(* IEC 61131-3 sources: CBasicModel/PLC/build, 2 files *)

(* ---- plc.st ---- *)
TYPE
  LOGLEVEL : (CRITICAL, WARNING, INFO, DEBUG) := INFO;
END_TYPE

FUNCTION_BLOCK LOGGER
  VAR_INPUT
    TRIG : BOOL;
    MSG : STRING;
    LEVEL : LOGLEVEL := INFO;
  END_VAR
  VAR
    TRIG0 : BOOL;
  END_VAR

  IF TRIG AND NOT TRIG0 THEN
  {{
   LogMessage(GetFbVar(LEVEL),(char*)GetFbVar(MSG, .body),GetFbVar(MSG, .len));
  }}
  END_IF;
  TRIG0:=TRIG;
END_FUNCTION_BLOCK

FUNCTION_BLOCK python_eval
  VAR_INPUT
    TRIG : BOOL;
    CODE : STRING;
  END_VAR
  VAR_OUTPUT
    ACK : BOOL;
    RESULT : STRING;
  END_VAR
  VAR
    STATE : DWORD;
    BUFFER : STRING;
    PREBUFFER : STRING;
    TRIGM1 : BOOL;
    TRIGGED : BOOL;
  END_VAR

  {extern void __PythonEvalFB(int, PYTHON_EVAL*);__PythonEvalFB(0, data__);}
END_FUNCTION_BLOCK

FUNCTION_BLOCK python_poll
  VAR_INPUT
    TRIG : BOOL;
    CODE : STRING;
  END_VAR
  VAR_OUTPUT
    ACK : BOOL;
    RESULT : STRING;
  END_VAR
  VAR
    STATE : DWORD;
    BUFFER : STRING;
    PREBUFFER : STRING;
    TRIGM1 : BOOL;
    TRIGGED : BOOL;
  END_VAR

  {extern void __PythonEvalFB(int, PYTHON_EVAL*);__PythonEvalFB(1,(PYTHON_EVAL*)(void*)data__);}
END_FUNCTION_BLOCK

FUNCTION_BLOCK python_gear
  VAR_INPUT
    N : UINT;
    TRIG : BOOL;
    CODE : STRING;
  END_VAR
  VAR_OUTPUT
    ACK : BOOL;
    RESULT : STRING;
  END_VAR
  VAR
    py_eval : python_eval;
    COUNTER : UINT;
    ADD10_OUT : UINT;
    EQ13_OUT : BOOL;
    SEL15_OUT : UINT;
    AND7_OUT : BOOL;
  END_VAR

  ADD10_OUT := ADD(COUNTER, 1);
  EQ13_OUT := EQ(N, ADD10_OUT);
  SEL15_OUT := SEL(EQ13_OUT, ADD10_OUT, 0);
  COUNTER := SEL15_OUT;
  AND7_OUT := AND(EQ13_OUT, TRIG);
  py_eval(TRIG := AND7_OUT, CODE := CODE);
  ACK := py_eval.ACK;
  RESULT := py_eval.RESULT;
END_FUNCTION_BLOCK

PROGRAM program0
  VAR
    PI_Taster_Links : BOOL;
    PI_LED_rot : BOOL;
    PI_LED_gruen : BOOL;
    PI_Taster_Rechts : BOOL;
    PI_LED_blau : BOOL;
    E_STOP : BOOL;
    E_Start : BOOL;
    E_Reset : BOOL;
    E_Hand_Automatik : BOOL;
    E_Links : BOOL;
    E_Rechts : BOOL;
    E_Drehmelder : BOOL;
    A_H1 : BOOL;
    A_H2 : BOOL;
    A_H3 : BOOL;
    A_H4 : BOOL;
    A_Motor_links : BOOL;
    A_Motor_rechts : BOOL;
    A_Motor_MaxSpeed : BOOL;
  END_VAR
  VAR
    NOT25_OUT : BOOL;
    NOT26_OUT : BOOL;
  END_VAR

  PI_LED_rot := E_Links;
  PI_LED_gruen := E_Rechts;
  NOT25_OUT := NOT(PI_Taster_Links);
  A_Motor_links := NOT25_OUT;
  NOT26_OUT := NOT(PI_Taster_Rechts);
  A_Motor_rechts := NOT26_OUT;
END_PROGRAM

CONFIGURATION Config0

  RESOURCE Res0 ON PLC
    TASK task0(INTERVAL := T#20ms,PRIORITY := 0);
    PROGRAM instance0 WITH task0 : program0;
  END_RESOURCE
END_CONFIGURATION

(* ---- generated_plc.st ---- *)
PROGRAM program0
  VAR
    PI_Taster_Links AT %IX0.0 : BOOL;
    PI_LED_rot AT %QX0.0 : BOOL;
    PI_LED_gruen AT %QX0.1 : BOOL;
    PI_Taster_Rechts AT %IX0.1 : BOOL;
    PI_LED_blau AT %QX0.2 : BOOL;
    E_STOP AT %QX4.0 : BOOL;
    E_Start AT %QX4.1 : BOOL;
    E_Reset AT %QX4.2 : BOOL;
    E_Hand_Automatik AT %QX4.3 : BOOL;
    E_Links AT %QX4.4 : BOOL;
    E_Rechts AT %QX4.5 : BOOL;
    E_Drehmelder AT %QX4.6 : BOOL;
    A_H1 AT %QX5.0 : BOOL;
    A_H2 AT %QX5.1 : BOOL;
    A_H3 AT %QX5.2 : BOOL;
    A_H4 AT %QX5.3 : BOOL;
    A_Motor_links AT %QX5.4 : BOOL;
    A_Motor_rechts AT %QX5.5 : BOOL;
    A_Motor_MaxSpeed AT %QX5.6 : BOOL;
  END_VAR
  VAR
    NOT25_OUT : BOOL;
    NOT26_OUT : BOOL;
  END_VAR

  PI_LED_rot := E_Links;
  PI_LED_gruen := E_Rechts;
  NOT25_OUT := NOT(PI_Taster_Links);
  A_Motor_links := NOT25_OUT;
  NOT26_OUT := NOT(PI_Taster_Rechts);
  A_Motor_rechts := NOT26_OUT;
END_PROGRAM

CONFIGURATION Config0

  RESOURCE Res0 ON PLC
    TASK task0(INTERVAL := T#20ms,PRIORITY := 0);
    PROGRAM instance0 WITH task0 : program0;
  END_RESOURCE
END_CONFIGURATION
